// TIA Portal V19 export
TYPE "PnDiag_Alr"
// stored: Access Published
   STRUCT
      Error : Bool;
      Module_Error : Bool;
   END_STRUCT;
END_TYPE
